{attribute 'qualified_only'}
{attribute 'strict'}
TYPE ActionMode :
(
	DoNothing	:= 0,
	AbsMove		:= 1,
	RelMove		:= 2,
	Home		:= 3,
	Find		:= 4
);
END_TYPE

(* stored: Version 1.1.0.1, ProductVersion 3.1.4024.15
   DUT ActionMode: Id {6f0fa8eb-32ee-4882-86a2-5afd36102fd1} *)
